INTERFACE I_ModuleServiceProperty

PROPERTY ModuleMode : T_PackMLMode
GET
END_GET
SET
END_SET
END_PROPERTY

END_INTERFACE

(* stored: Version 1.1.0.1, ProductVersion 3.1.4026.18
   Itf I_ModuleServiceProperty: Id {b0c61b72-0d64-4968-b250-19f75305f691}
   Property ModuleMode: Id {ec976903-4c6f-49fb-927f-d95c2422c8ab}
   Get Get: Id {94527eed-53c7-4795-a31e-2c4291402721}
   Set Set: Id {ff21a37e-a437-4d73-98f0-b2191ccfb9db} *)
